INTERFACE I_PersistentEventStorage

METHOD StoreEvent
VAR_INPUT
	stEvent	:	ST_Event;
END_VAR
END_METHOD

END_INTERFACE

(* stored: Version 1.1.0.1, ProductVersion 3.1.4024.12
   Itf I_PersistentEventStorage: Id {a50ac1f9-778b-43cf-a6bb-8d175462cdab}
   Method StoreEvent: Id {327bf44c-be19-4d30-8f80-233817c2dfb8} *)
